{attribute 'linkalways'} 
{attribute 'no_explicit_call' := 'This FB is a CLASS and must be accessed using methods or properties'}
{attribute 'enable_dynamic_creation'}
FUNCTION_BLOCK _UINT EXTENDS NumericDatatypeBase
VAR
	localData : UINT;
	activeData : REFERENCE TO UINT REF= localData;
END_VAR

PROPERTY PUBLIC Address : PVOID
GET
Address := ADR(activeData);
END_GET
END_PROPERTY

METHOD PUBLIC ClearReference
VAR_INPUT
END_VAR
activeData REF= localData;
END_METHOD

METHOD PUBLIC Clone : I_Datatype
VAR
    pClone : POINTER TO _UINT;
END_VAR
pClone := __NEW(_UINT(InitialValue := Value));
Clone := pClone^;
END_METHOD

METHOD FB_init : BOOL
VAR_INPUT
	bInitRetains : BOOL; // if TRUE, the retain variables are initialized (warm start / cold start)
	bInCopyCode : BOOL;  // if TRUE, the instance afterwards gets moved into the copy code (online change)
	InitialValue : UINT;
END_VAR
localData := InitialValue;
END_METHOD

PROPERTY PUBLIC IsEven : BOOL
GET
IsEven := (Value mod 2) = 0;
END_GET
END_PROPERTY

PROPERTY PUBLIC IsFloat : BOOL
GET
IsFloat := FALSE;
END_GET
END_PROPERTY

PROPERTY PUBLIC IsSigned : BOOL
GET
IsSigned := FALSE;
END_GET
END_PROPERTY

METHOD PUBLIC MakeReferenceTo
VAR_INPUT
	ReferenceTarget : REFERENCE TO UINT;
END_VAR
activeData REF= ReferenceTarget;
END_METHOD

PROPERTY PUBLIC MaxValue : UINT
GET
MaxValue :=  DatatypeLimits.UINT_MAX_VALUE;
END_GET
END_PROPERTY

PROPERTY PUBLIC MinValue : UINT
GET
MinValue := DatatypeLimits.UINT_MIN_VALUE;
END_GET
END_PROPERTY

METHOD PROTECTED SerializeMaxValue
VAR_INPUT
	Serializer : I_Serializer;
END_VAR
Serializer.AddUint(MaxValue);
END_METHOD

METHOD PROTECTED SerializeMinValue
VAR_INPUT
	Serializer : I_Serializer;
END_VAR
Serializer.AddUint(MinValue);
END_METHOD

METHOD PUBLIC SerializeWith
VAR_INPUT
	Serializer : I_Serializer;
END_VAR
Serializer.AddUint(activeData);
END_METHOD

PROPERTY PUBLIC Size : UDINT
GET
Size := SIZEOF(activeData);
END_GET
END_PROPERTY

METHOD TryDeserializeFrom : BOOL
VAR_INPUT
	Deserializer : I_Deserializer;
	Feedback : I_DeserializerFeedback;
END_VAR
TryDeserializeFrom := Deserializer.TryGetUint(activeData, Feedback);
END_METHOD

METHOD TryMakeReferenceTo : BOOL
VAR_INPUT
	Target : I_Datatype;
END_VAR
VAR
	pTargetData : POINTER TO UINT;
END_VAR
IF NOT (Target.TypeName = TypeName) THEN
	RETURN;
END_IF

pTargetData := Target.Address;
activeData REF= pTargetData^;
TryMakeReferenceTo := TRUE;
END_METHOD

PROPERTY PUBLIC TypeName : T_MAXSTRING
GET
TypeName := 'UINT';
END_GET
END_PROPERTY

PROPERTY PUBLIC Value : REFERENCE TO UINT
GET
Value REF= activeData;
END_GET
END_PROPERTY

END_FUNCTION_BLOCK

(* stored: Version 1.1.0.1, ProductVersion 3.1.4024.13
   POU _UINT: Id {db5ef119-9b74-4fad-aee9-d04bb2ab64dc}, SpecialFunc None
   Folder Constructor: Id {3aa93293-a1d0-4b15-abea-25b00ada61b0}
   Folder Protected: Id {17a4be64-c0c7-4fe2-869c-44d3a2d114d4}
   Property Address: Id {d3107168-cea2-4a6e-bfc7-f4d56dea99e1}
   Get Get: Id {5564fe73-0ca4-48f3-bcb1-907a209b5aed}
   Method ClearReference: Id {d982472e-1368-4245-a2ac-a887ac368e5a}
   Method Clone: Id {8afe84e2-9b30-4836-9429-d5ede9998bb2}
   Method FB_init: Id {593e5964-57c3-481c-a2bb-66af58015659}
   Property IsEven: Id {60974194-023b-0e6f-2dee-abbbac23a692}
   Get Get: Id {439ac2b9-9b13-0b63-2b16-fc9d0e7bd569}
   Property IsFloat: Id {3343f0b9-d57b-4fcb-b19f-eabc293d7b5c}
   Get Get: Id {be640483-5dcb-42c8-9690-d23c7689593d}
   Property IsSigned: Id {7ff70222-b5d6-4e9c-9729-8bbed37bfe59}
   Get Get: Id {d503bb5e-9ccd-4c78-b365-fc9ad9b9f7fd}
   Method MakeReferenceTo: Id {f301e36b-870b-4ede-8106-3e45a008dfce}
   Property MaxValue: Id {45091765-df0a-4e66-a0f8-e18862a9888c}
   Get Get: Id {1e05c93c-388f-4b18-9aa2-b0cfb17840c4}
   Property MinValue: Id {23a5e76e-0c4c-4626-a3ae-29670238ebfd}
   Get Get: Id {5bec5776-d1ec-43f9-aeb0-046dc3800e96}
   Method SerializeMaxValue: Id {7321e6af-fe15-42d6-ab68-57b1e56e9cba}
   Method SerializeMinValue: Id {9aaae453-c4c0-453d-bdd4-7930aef2e599}
   Method SerializeWith: Id {0b49458e-e9ea-4020-afcc-154c4733d6ae}
   Property Size: Id {fdb97a21-b5e9-4865-aafb-e89aae81481b}
   Get Get: Id {0518eb7b-dd1c-4781-a30b-53dcf423ac33}
   Method TryDeserializeFrom: Id {a1b3b02a-6503-4e89-b5e1-9bdd3e477a99}
   Method TryMakeReferenceTo: Id {a0883963-8dfd-46f6-9d04-d03dea66477c}
   Property TypeName: Id {d676e6b2-49ed-4692-a8d6-329bd2466efc}
   Get Get: Id {730428a8-cba6-47b0-ab3d-5655a04b17b1}
   Property Value: Id {f3f0c4a3-be7e-49de-b4da-2a398a3e11f7}
   Get Get: Id {ecf19aa1-532d-4bb7-afa2-ffaded59098c} *)
